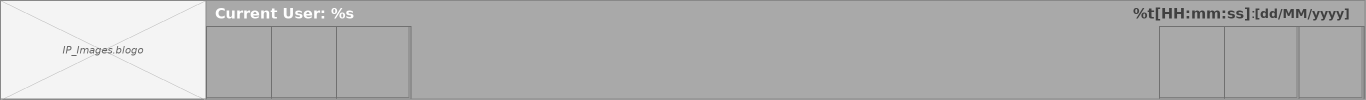
VISUALIZATION PH_Header  // 1366x100
VAR_IN_OUT
	iFrameNumber							: INT;
	bMenu 									: BOOL;
	wButton									: WORD;
END_VAR
    Button (211,34 65x65), image: IP_Buttons.menu dark
        OnMouseEnter: execute { GVL_HMI.wButton.0:=TRUE; }
        OnMouseLeave: execute { GVL_HMI.wButton.0:=FALSE; }
        OnMouseDown: execute { GVL_HMI.bMenu:=TRUE; }
    Rectangle (1233,1 120x25), "%t[dd/MM/yyyy]"
    Rectangle (212,1 250x25), "Current User: %s", text variable: VisuElemsWinControls.CurrentFullUserName
    Button (276,34 65x65), image: IP_Buttons.home dark
        OnMouseEnter: execute { GVL_HMI.wButton.1:=TRUE; }
        OnMouseLeave: execute { GVL_HMI.wButton.1:=FALSE; }
        OnMouseDown: execute { GVL_HMI.iFrameNumber:=0; GVL_HMI.bMenu:=FALSE; }
    Button (341,34 65x65), image: IP_Buttons.alarms dark
        OnMouseEnter: execute { GVL_HMI.wButton.2:=TRUE; }
        OnMouseLeave: execute { GVL_HMI.wButton.2:=False; }
        OnMouseDown: execute { GVL_HMI.iFrameNumber:=1; GVL_HMI.bMenu:=FALSE; }
    Button (1164,34 65x65), image: IP_Buttons.info dark
        OnMouseEnter: execute { GVL_HMI.wButton.3:=TRUE; }
        OnMouseLeave: execute { GVL_HMI.wButton.3:=FALSE; }
        OnMouseDown: execute { GVL_HMI.iFrameNumber:=2; GVL_HMI.bMenu:=FALSE; }
    Button (1229,34 65x65), colour toggle: GVL_HMI.wButton.4, image: IP_Buttons.user dark
        OnMouseEnter: execute { GVL_HMI.wButton.4:=TRUE; }
        OnMouseLeave: execute { GVL_HMI.wButton.4:=FALSE; }
        OnMouseDown: execute { GVL_HMI.iFrameNumber:=3; GVL_HMI.bMenu:=FALSE; }
    Button (1294,34 65x65), image: IP_Buttons.set dark
        OnMouseEnter: execute { GVL_HMI.wButton.5:=TRUE; }
        OnMouseLeave: execute { GVL_HMI.wButton.5:=FALSE; }
        OnMouseDown: execute { GVL_HMI.iFrameNumber:=4; GVL_HMI.bMenu:=FALSE; }
    Rectangle (1132,1 120x25), "%t[HH:mm:ss]"
    RoundedRectangle (625,53 280x40), text list: 'TL_Frames', text index: iFrameNumber
    Image (0,0 206x100), image: IP_Images.blogo
    Button (1229,34 65x65), invisible if: NOT GVL_HMI.wButton.4, image: IP_Buttons.user light
        OnMouseEnter: execute { GVL_HMI.wButton.4:=TRUE; }
        OnMouseLeave: execute { GVL_HMI.wButton.4:=FALSE; }
        OnMouseDown: execute { GVL_HMI.iFrameNumber:=3; GVL_HMI.bMenu:=FALSE; }
    Button (1294,34 65x65), invisible if: NOT GVL_HMI.wButton.5, image: IP_Buttons.set light
        OnMouseEnter: execute { GVL_HMI.wButton.5:=TRUE; }
        OnMouseLeave: execute { GVL_HMI.wButton.5:=FALSE; }
        OnMouseDown: execute { GVL_HMI.iFrameNumber:=4; GVL_HMI.bMenu:=FALSE; }
    Button (1289,26 75x73), invisible if: iFrameNumber<>4 OR GVL_HMI.bMenu, image: IP_Buttons.set dark
        OnMouseEnter: execute { GVL_Hmi.wButton.5:=TRUE; }
        OnMouseLeave: execute { GVL_Hmi.wButton.5:=FALSE; }
    Button (1289,26 75x73), invisible if: iFrameNumber<>4 OR GVL_HMI.bMenu OR NOT GVL_HMI.wButton.5, image: IP_Buttons.set light
        OnMouseEnter: execute { GVL_Hmi.wButton.5:=TRUE; }
        OnMouseLeave: execute { GVL_Hmi.wButton.5:=FALSE; }
    Button (1164,34 65x65), invisible if: NOT GVL_HMI.wButton.3, image: IP_Buttons.info light
        OnMouseEnter: execute { GVL_HMI.wButton.3:=TRUE; }
        OnMouseLeave: execute { GVL_HMI.wButton.3:=FALSE; }
        OnMouseDown: execute { GVL_HMI.iFrameNumber:=2; GVL_HMI.bMenu:=FALSE; }
    Button (1159,26 75x73), invisible if: iFrameNumber<>2 OR GVL_HMI.bMenu, image: IP_Buttons.info dark
        OnMouseEnter: execute { GVL_Hmi.wButton.3:=TRUE; }
        OnMouseLeave: execute { GVL_Hmi.wButton.3:=FALSE; }
    Button (1159,26 75x73), invisible if: iFrameNumber<>2 OR GVL_HMI.bMenu OR NOT GVL_HMI.wButton.3, image: IP_Buttons.info light
        OnMouseEnter: execute { GVL_Hmi.wButton.3:=TRUE; }
        OnMouseLeave: execute { GVL_Hmi.wButton.3:=FALSE; }
    Button (341,34 65x65), invisible if: NOT GVL_HMI.wButton.2, image: IP_Buttons.alarms light
        OnMouseEnter: execute { GVL_HMI.wButton.2:=TRUE; }
        OnMouseLeave: execute { GVL_HMI.wButton.2:=False; }
        OnMouseDown: execute { GVL_HMI.iFrameNumber:=1; GVL_HMI.bMenu:=FALSE; }
    Button (276,34 65x65), invisible if: NOT GVL_HMI.wButton.1, image: IP_Buttons.home light
        OnMouseEnter: execute { GVL_HMI.wButton.1:=TRUE; }
        OnMouseLeave: execute { GVL_HMI.wButton.1:=FALSE; }
        OnMouseDown: execute { GVL_HMI.iFrameNumber:=0; GVL_HMI.bMenu:=FALSE; }
    Button (1224,26 75x73), invisible if: iFrameNumber<>3 OR GVL_HMI.bMenu, image: IP_Buttons.user dark
        OnMouseEnter: execute { GVL_Hmi.wButton.4:=TRUE; }
        OnMouseLeave: execute { GVL_Hmi.wButton.4:=FALSE; }
    Button (1224,26 75x73), invisible if: iFrameNumber<>3 OR GVL_HMI.bMenu OR NOT GVL_HMI.wButton.4, image: IP_Buttons.user light
        OnMouseEnter: execute { GVL_Hmi.wButton.4:=TRUE; }
        OnMouseLeave: execute { GVL_Hmi.wButton.4:=FALSE; }
    Button (211,34 65x65), invisible if: NOT GVL_HMI.wButton.0, image: IP_Buttons.menu light
        OnMouseEnter: execute { GVL_HMI.wButton.0:=TRUE; }
        OnMouseLeave: execute { GVL_HMI.wButton.0:=FALSE; }
        OnMouseDown: execute { GVL_HMI.bMenu:=TRUE; }
    Button (206,26 75x73), invisible if: NOT GVL_HMI.bMenu, image: IP_Buttons.menu dark
        OnMouseEnter: execute { GVL_Hmi.wButton.0:=TRUE; }
        OnMouseLeave: execute { GVL_Hmi.wButton.0:=FALSE; }
    Button (206,26 75x73), invisible if: NOT GVL_HMI.bMenu OR NOT GVL_HMI.wButton.0, image: IP_Buttons.menu light
        OnMouseEnter: execute { GVL_Hmi.wButton.0:=TRUE; }
        OnMouseLeave: execute { GVL_Hmi.wButton.0:=FALSE; }
    Button (271,26 75x73), invisible if: iFrameNumber<>0 OR GVL_HMI.bMenu, image: IP_Buttons.home dark
        OnMouseEnter: execute { GVL_Hmi.wButton.1:=TRUE; }
        OnMouseLeave: execute { GVL_Hmi.wButton.1:=FALSE; }
    Button (271,26 75x73), invisible if: iFrameNumber<>0 OR GVL_HMI.bMenu OR NOT GVL_HMI.wButton.1, image: IP_Buttons.home light
        OnMouseEnter: execute { GVL_Hmi.wButton.1:=TRUE; }
        OnMouseLeave: execute { GVL_Hmi.wButton.1:=FALSE; }
    Button (336,26 75x73), invisible if: iFrameNumber<>1 OR GVL_HMI.bMenu, image: IP_Buttons.alarms dark
        OnMouseEnter: execute { GVL_Hmi.wButton.2:=TRUE; }
        OnMouseLeave: execute { GVL_Hmi.wButton.2:=FALSE; }
    Button (336,26 75x73), invisible if: iFrameNumber<>1 OR GVL_HMI.bMenu OR NOT GVL_HMI.wButton.2, image: IP_Buttons.alarms light
        OnMouseEnter: execute { GVL_Hmi.wButton.2:=TRUE; }
        OnMouseLeave: execute { GVL_Hmi.wButton.2:=FALSE; }
END_VISUALIZATION

(* stored: Version 1.1.0.1, ProductVersion 3.1.4024.3
   Visu PH_Header: Id {f764203b-540a-4159-8103-5cd882ab5fee} *)
